// TIA Portal V18 export
FUNCTION "Block_LADDER" : Void   // FC5, LAD
{ S7_Optimized_Access := 'TRUE' }
VERSION : 0.1
// stored: AutoNumber true, IsIECCheckEnabled false, SetENOAutomatically false, UDAEnableTagReadback false
BEGIN

REGION Network 1
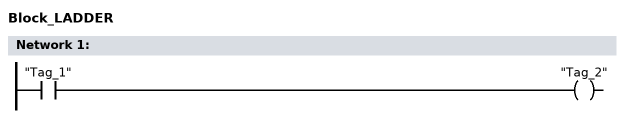
   RUNG wire#powerrail
      Contact( "Tag_1" )
      Coil( "Tag_2" )
   END_RUNG
   // the same network as SCL:
   "Tag_2" := "Tag_1";
END_REGION
END_FUNCTION
